Fanuc KAREL source: kb00077.KL

PROGRAM KB00077
%NOLOCKGROUP
VAR
P1 : STRING[80];P2:INTEGER;P3:INTEGER;P4 : STRING[80];P5:INTEGER
BEGIN
--
--
--
--
P1='A'
P2=1
P3=1
P4='A'
P5=1
GET_ATTR_PRG(P1,P2,P3,P4,P5)
END KB00077
